% RSLogix 500 project Project_6.RSS, saved by version 8.30.00.16 %
PROJECT "UNTITLED"    % processor: Bul.1763 MicroLogix 1100 Series B %

PROGRAM FILES
  LAD 2   3 rungs
  LAD 3 "IO"  3 rungs
  LAD 4 "CONTROL"  7 rungs

DATA FILES
  O0 OUTPUT  5 elements
  I1 INPUT  7 elements
  S2 STATUS  66 elements
  B3 BINARY  3 elements
  T4 TIMER  1 elements
  C5 COUNTER  3 elements
  R6 CONTROL  1 elements
  N7 INTEGER  4 elements
  F8 FLOAT  1 elements

LADDER 2
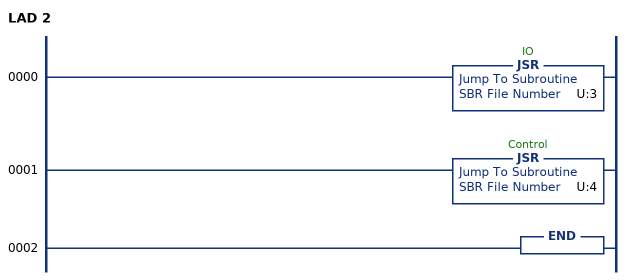
% Rung: 0 %
SOR JSR U:3 EOR
%   U:3  "IO" %
% Rung: 1 %
SOR JSR U:4 EOR
%   U:4  "Control" %
% Rung: 2 %
SOR END EOR

LADDER 3 "IO"
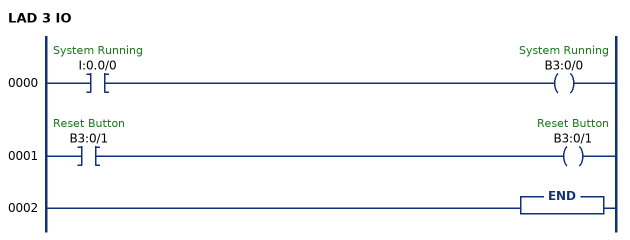
% Rung: 0 %
SOR XIC I:0.0/0 OTE B3:0/0 EOR
%   I:0.0/0  "System Running" %
%   B3:0/0  "System Running" %
% Rung: 1 %
SOR XIC B3:0/1 OTE B3:0/1 EOR
%   B3:0/1  "Reset Button" %
% Rung: 2 %
SOR END EOR

LADDER 4 "CONTROL"
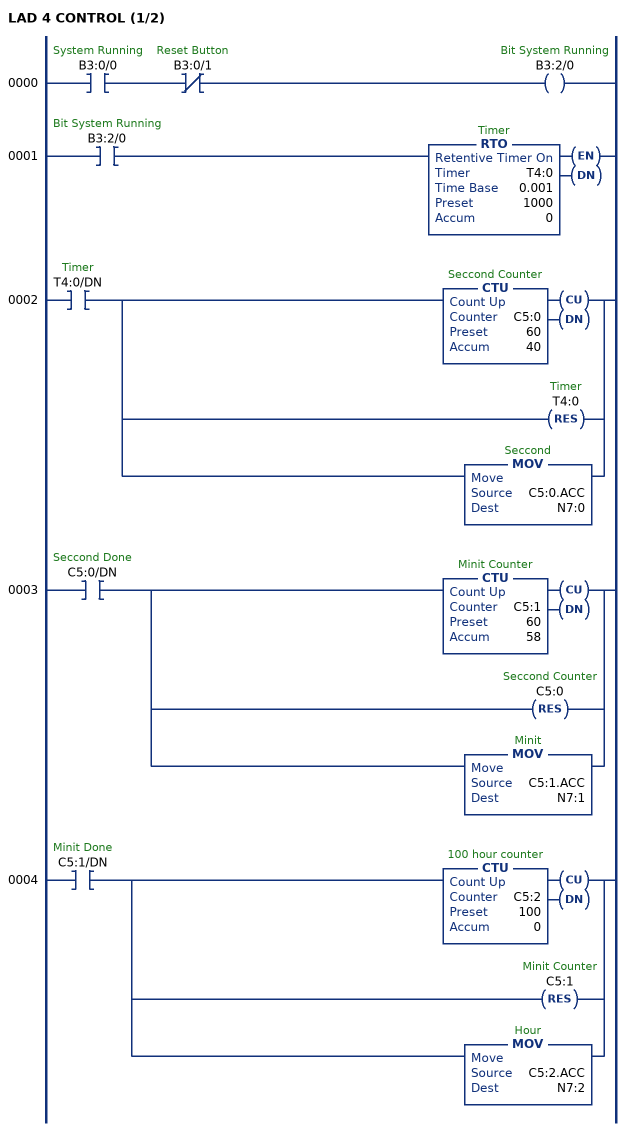
% Rung: 0 %
SOR XIC B3:0/0 XIO B3:0/1 OTE B3:2/0 EOR
%   B3:0/0  "System Running" %
%   B3:0/1  "Reset Button" %
%   B3:2/0  "Bit System Running" %
% Rung: 1 %
SOR XIC B3:2/0 RTO T4:0 0.001 1000 0 EOR
%   B3:2/0  "Bit System Running" %
%   T4:0  "Timer" %
% Rung: 2 %
SOR XIC T4:0/DN BST CTU C5:0 60 40 NXB RES T4:0 NXB MOV C5:0.ACC N7:0 BND EOR
%   T4:0  "Timer" %
%   C5:0  "Seccond Counter" %
%   C5:0.ACC  "Seccond" %
%   N7:0  "Seccond" %
% Rung: 3 %
SOR XIC C5:0/DN BST CTU C5:1 60 58 NXB RES C5:0 NXB MOV C5:1.ACC N7:1 BND EOR
%   C5:0/DN  "Seccond Done" %
%   C5:1  "Minit Counter" %
%   C5:0  "Seccond Counter" %
%   C5:1.ACC  "Minit" %
%   N7:1  "Minit" %
% Rung: 4 %
SOR XIC C5:1/DN BST CTU C5:2 100 0 NXB RES C5:1 NXB MOV C5:2.ACC N7:2 BND EOR
%   C5:1/DN  "Minit Done" %
%   C5:2  "100 hour counter" %
%   C5:1  "Minit Counter" %
%   C5:2.ACC  "Hour" %
%   N7:2  "Hour" %

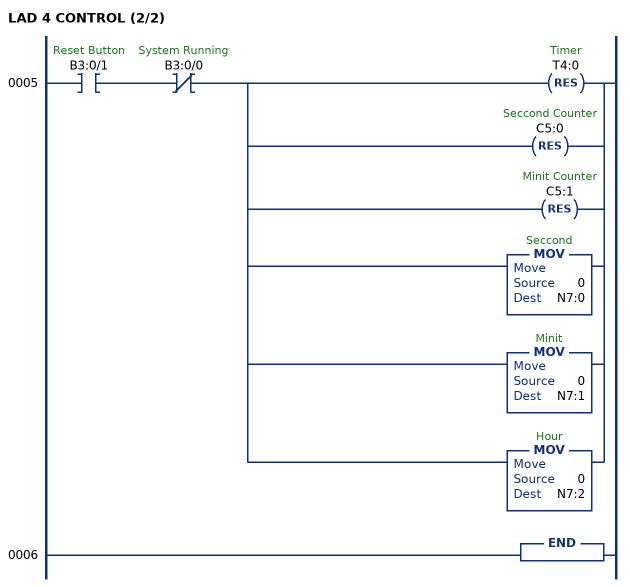
% Rung: 5 %
SOR XIC B3:0/1 XIO B3:0/0 BST RES T4:0 NXB RES C5:0 NXB RES C5:1 NXB MOV 0 N7:0 NXB MOV 0 N7:1 NXB MOV 0 N7:2 BND EOR
%   B3:0/1  "Reset Button" %
%   B3:0/0  "System Running" %
%   T4:0  "Timer" %
%   C5:0  "Seccond Counter" %
%   C5:1  "Minit Counter" %
%   N7:0  "Seccond" %
%   N7:1  "Minit" %
%   N7:2  "Hour" %
% Rung: 6 %
SOR END EOR

OTHER DOCUMENTED ADDRESSES
  B3:1/0  "ONS"
  I:0.0/2  "Reset Button"
  T4:1  "Minit"

DATA TABLE (non-zero values as saved)
DATA T4
% .PRE .ACC %
% T4:0 % 1000 0
DATA C5
% .PRE .ACC %
% C5:0 % 60 40
% C5:1 % 60 58
% C5:2 % 100 0
